FUNCTION_BLOCK earth_fault_1_2_backup (* Composite Function Block Type *)
  (* Standard: 61499-2 *)
  (* Version 0.0, 3/23/2016, gulzha, nxtControl GmbH, template *)
  PACKAGE Main;
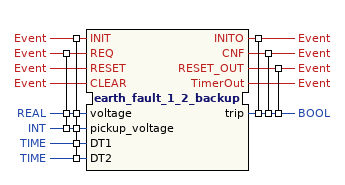
  EVENT_INPUT
    INIT WITH pickup_voltage, voltage, DT1, DT2; (* Initialization Request *)
    REQ WITH pickup_voltage, voltage; (* Normal Execution Request *)
    RESET;
    CLEAR;
  END_EVENT
  EVENT_OUTPUT
    INITO WITH trip; (* Initialization Confirm *)
    CNF WITH trip; (* Execution Confirmation *)
    RESET_OUT WITH trip;
    TimerOut;
  END_EVENT
  VAR_INPUT
    voltage : REAL;
    pickup_voltage : INT;
    DT1 : TIME; (* Delay Time *)
    DT2 : TIME; (* Delay Time *)
  END_VAR
  VAR_OUTPUT
    trip : BOOL;
  END_VAR
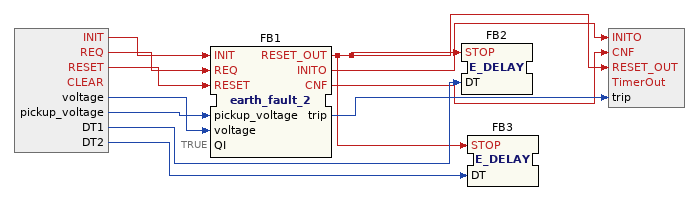
  FBS
    FB2 : E_DELAY;
    FB3 : E_DELAY;
    FB1 : earth_fault_2(QI := TRUE);
  END_FBS
  EVENT_CONNECTIONS
    FB1.RESET_OUT TO FB2.STOP;
    FB1.RESET_OUT TO FB3.STOP;
    INIT TO FB1.INIT;
    FB1.INITO TO INITO;
    REQ TO FB1.REQ;
    RESET TO FB1.RESET;
    FB1.RESET_OUT TO RESET_OUT;
    FB1.CNF TO CNF;
  END_CONNECTIONS
  DATA_CONNECTIONS
    pickup_voltage TO FB1.pickup_voltage;
    voltage TO FB1.voltage;
    FB1.trip TO trip;
    DT1 TO FB2.DT;
    DT2 TO FB3.DT;
  END_CONNECTIONS
END_FUNCTION_BLOCK
